TYPE SPEED_CORRECTION_PERCENT : SINT(IntersectionConstants.MIN_LIGHT_SWITCH_SPEED_CORECTION_PERCENT..IntersectionConstants.MAX_LIGHT_SWITCH_SPEED_CORECTION_PERCENT); END_TYPE

(* stored: Version 1.1.0.1
   DUT SPEED_CORRECTION_PERCENT: Id {6eaae858-42d0-488e-8e43-0349f96f99f9} *)
